// TIA Portal V20 export
ORGANIZATION_BLOCK "CyclicInterrupt"   // OB30, LAD, CyclicInterrupt
{ S7_Optimized_Access := 'TRUE' }
// stored: SetENOAutomatically false
   VAR_INPUT
      Initial_Call : Bool;   // Initial call of this OB
      Event_Count : Int;   // Events discarded
   END_VAR
BEGIN

REGION Network 2
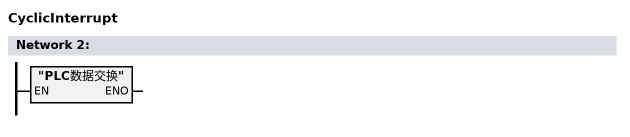
   RUNG wire#powerrail
      "PLC数据交换"()
   END_RUNG
   // the same network as SCL:
   "PLC数据交换"();
END_REGION
END_ORGANIZATION_BLOCK
